FUNCTION HPF_Function : REAL
VAR_INPUT
	SignalToFilter : REAL;
	FilterParams : POINTER TO HighPassFilter;
END_VAR
VAR
END_VAR

HPF_Function := FilterParams^.b0*SignalToFilter + FilterParams^.b1*FilterParams^.ErrorFilt - FilterParams^.a1*Filterparams^.OutputFilt;

FilterParams^.ErrorFilt := SignalToFilter;
FilterParams^.OutputFilt := HPF_Function;

END_FUNCTION

(* stored: Version 1.1.0.1, ProductVersion 3.1.4024.4
   POU HPF_Function: Id {d425d246-1428-4be6-8a8e-dca788ef7830}, SpecialFunc None *)
